Fanuc TP program (LS listing): _LOG_TEST.LS

/PROG  _LOG_TEST
/ATTR
OWNER		= MNEDITOR;
COMMENT		= "";
PROG_SIZE	= 215;
CREATE		= DATE 21-05-20  TIME 13:16:32;
MODIFIED	= DATE 21-05-20  TIME 13:17:06;
FILE_NAME	= ;
VERSION		= 0;
LINE_COUNT	= 1;
MEMORY_SIZE	= 591;
PROTECT		= READ_WRITE;
TCD:  STACK_SIZE	= 0,
      TASK_PRIORITY	= 50,
      TIME_SLICE	= 0,
      BUSY_LAMP_OFF	= 0,
      ABORT_REQUEST	= 0,
      PAUSE_REQUEST	= 0;
DEFAULT_GROUP	= 1,*,*,*,*;
CONTROL_CODE	= 00000000 00000000;
/APPL
/APPL

AUTO_SINGULARITY_HEADER;
  ENABLE_SINGULARITY_AVOIDANCE   : TRUE;

  AUTOZONE_INTERFERENCE_AVOID;
    AUTOZONE_ENABLED         : FALSE;
    AUTOZONE_SCHEDULE_NUMBER : 1;
/MN
   1:  CALL KL_LOGGER_TEST    ;
/POS
/END
